TYPE E_ModalGeoTypes :
(
	MODALGEOTYPE_Undefined := 0,
	MODALGEOTYPE_G0 := 4096,
	MODALGEOTYPE_G01 := 4097,
	MODALGEOTYPE_G02 := 4098,
	MODALGEOTYPE_G03 := 4099
)UDINT;
END_TYPE

(* stored: Version 1.1.0.1, ProductVersion 3.1.0.25
   DUT E_ModalGeoTypes: Id {8737441b-d59d-4e79-9915-d37b409b501d} *)
